{attribute 'qualified_only'}
TYPE E_SDSGarageYStates :
(
    UNKNOWN := 0,
    T1 := 1,
    T2 := 2,
    T3 := 3,
    T4 := 4,
    M1 := 5,
    M2 := 6,
    M3 := 7,
    M4 := 8,
    B1 := 9,
    B2 := 10,
    B3 := 11,
    B4 := 12,
    RETRACTED := 13
) UINT;
END_TYPE

(* stored: Version 1.1.0.1
   DUT E_SDSGarageYStates: Id {1c493091-840f-4f55-aa53-dd2a7692158f} *)
